TYPE ST_GenericHierarchy_Write :
STRUCT
	HierarchyType		:STRING;
	_ACTION				:STRING;
	TrackingLevels		:STRING;
	TrackingIndicator	:STRING;
	ItemCS				:ST_ItemCS;
END_STRUCT
END_TYPE

(* stored: Version 1.1.0.1, ProductVersion 3.1.4024.13
   DUT ST_GenericHierarchy_Write: Id {f3f12d3d-3765-4f29-89c4-b2f6495b8771} *)
